(* IEC 61131-3 sources: Nauka-PLC-ST/ (part 2) *)

(* ---- Sterownik_Prasy_Formujacej.st ---- *)
VAR
    Start : BOOL;           // Przycisk monostabilny (musi być trzymany)
    Czujnik_detalu : BOOL;  // Potwierdzenie obecności materiału
    Czujnik_gora : BOOL;    // Czujnik prasy w gornym polozeniu
    Czujnik_dol : BOOL;     // Czujnik prasyw dolnym polozeniu
    Zawor_3_2 : BOOL;       // 1 - wysunięcie, 0 - schowanie (sprężyna)
    Krok_ukladu : INT := 0;
    Timer_prasowania : TON;
END_VAR

Timer_prasowania(PT := T#5S);

CASE Krok_ukladu OF
    0:  // IDLE - Czekamy na start i detal
        Zawor_3_2 := FALSE;
        Timer_prasowania.IN := FALSE;

        IF Start AND Czujnik_detalu THEN
            Krok_ukladu := 1;
        END_IF;

    1:  // ruch silownika w dol
        IF Start THEN
            Zawor_3_2 := TRUE;
            IF Czujnik_dol THEN // pzrechodzimy dopiero gdy silownik zjedzie na dol
                Krok_ukladu := 2;
            END_IF;
        ELSE
            // silownik wraca gdy puszcze przycisk start
            Krok_ukladu := 0;
        END_IF;

    2:  // czas pasowania detalu
        IF Start THEN
            Zawor_3_2 := TRUE;
            Timer_prasowania.IN := TRUE; // timer odlicza czas

            IF Timer_prasowania.Q THEN
                Krok_ukladu := 3;
            END_IF;
        ELSE
            Krok_ukladu := 0; // przerwanie prasowania
        END_IF;

    3:  // powrot silownika do stanu poczatkowego
        Zawor_3_2 := FALSE;
        Timer_prasowania.IN := FALSE;

        // Czekamy chwilę aż siłownik wróci (można dodać czujnik góra)
        IF NOT Start AND Czujnik_gora THEN
            Krok_ukladu := 0;
        END_IF;
END_CASE;

(* ---- Sterownik_przedmuchu_filtrow.st ---- *)
VAR
    Presostat_roznicy_p  : BOOL;  // czujnik przekroczenia max roznicy cisnien - filtr zapchany
    Zezwolenie_pracy     : BOOL;  // sygnal potwierdzajacy prace wlownego wentylatora

    Timer_impulsu        : TON;   // timer kontrolujacy czas trwania strzalu powietrza (np. 500ms)
    Timer_pauzy          : TON;   // timer liczacy przerwe miedzy strzalami roznych sekcji
    Krok                 : INT;   // krok ukladu: 0-spoczynek, 1-strzal 1, 2-pauza, 3-strzal 2

    Zawor_Przedmuchu_1   : BOOL;  // elektrozawor sprzonego powietrza dla sekcji 1
    Zawor_Przedmuchu_2   : BOOL;  // elektrozawor sprzonego powietrza dla sekcji 2
END_VAR

CASE Krok OF
    0: // Oczekiwanie na sygnal zapchania filtra przy pracy
        IF Presostat_roznicy_p AND Zezwolenie_pracy THEN
            Krok := 1; // rozpoczecie regeneracji
        END_IF;

    1: // strzal powietrza - sekcja 1
        IF Timer_impulsu.Q THEN
            Krok := 2; // koniec strzalu -> przejdz do pauzy
        END_IF;

    2: // przerwa na powrot cisnienia w zbiorniku
        IF Timer_pauzy.Q THEN
            Krok := 3; // powrot cisnienia -> strzal na sekcje 2
        END_IF;

    3: // Strzal powietrza - sekcja 2
        IF Timer_impulsu.Q THEN
            Krok := 0; // koniec oczyszczania -> powrot do czuwania
        END_IF;
END_CASE;

// timery
Timer_impulsu(IN := (Krok = 1) OR (Krok = 3), PT := T#500ms);  // czas pojedynczego strzalu powietrza

Timer_pauzy(IN := (Krok = 2), PT := T#4s);  // czas powrotu cisnienia

// sterowanie wyjsciami
Zawor_Przedmuchu_1 := Zezwolenie_pracy AND (Krok = 1);
Zawor_Przedmuchu_2 := Zezwolenie_pracy AND (Krok = 3);

(* ---- Sterownik_rozladunku_silosu.st ---- *)
VAR
    Zadanie_rozladunku   : BOOL;  // sygnal zadania startusekwencji programu
    Czujnik_przeplywu    : BOOL;  // czujnik lub fotokomorka wykrywajacy fizyczny zrzut materialu
    Krancowka_zasuwy     : BOOL;  // potwierdzenie pelnego otwarcia zasuwy pod silosem

    Timer_aeracji        : TON;   // czas trwania strzalu powietrza
    Timer_wibracji       : TON;   // czas pracy wibratora
    Krok                 : INT;   // krok sekwencji

    Zasuwa_nozowa        : BOOL;  // otwarcie zasuwy odcinajacej silos
    Zawor_aeracji        : BOOL;  // cewka elektrozaworu wtrysku powietrza
    Wibrator_stozka      : BOOL;  // stycznik silnika wibracyjnego na plaszczu
END_VAR

CASE Krok OF
    0: // stan czuwania - oczekiwanie na rozpoczecie sekwencji
        IF Zadanie_rozladunku THEN
            Krok := 1; // rozpoczecie rozladunku
        END_IF;

    1: // standardowy zrzut po otwarciu zrzutu
        IF NOT Zadanie_rozladunku THEN
            Krok := 0; // koniec rozladunku
        ELSIF Zadanie_rozladunku AND NOT Czujnik_przeplywu AND Krancowka_zasuwy THEN
            Krok := 2; // otawrta zasuwa - wykryto zwis
        END_IF;

    2: // spulchnianie materialu
        IF NOT Zadanie_rozladunku THEN
            Krok := 0;
        ELSIF Timer_aeracji.Q THEN
            IF Czujnik_przeplywu THEN
                Krok := 1; // powrot do standardowego zrzutu
            ELSE
                Krok := 3; // przejscie do wibracji
            END_IF;
        END_IF;

    3: // aktwyacja wibratora
        IF NOT Zadanie_rozladunku OR Timer_wibracji.Q OR Czujnik_przeplywu THEN
            Krok := 1; // powrot do oczekiwanie na rozpoczecie nowej sekwencji
        END_IF;
END_CASE;

// timer

Timer_aeracji(IN := (Krok = 2), PT := T#4s); // strzal powietrz trwa 4 sekundy

// Praca wibratora ograniczona do 3 sekund, aby chronic strukture mechaniczna i spawy silosu
Timer_wibracji(IN := (Krok = 3), PT := T#3s);

// sterowanie wyjsciami
Zasuwa_nozowa   := (Krok = 1) OR (Krok = 2) OR (Krok = 3);
Zawor_aeracji   := (Krok = 2);
Wibrator_stozka := (Krok = 3);

(* ---- Sterownik_stacji_obrotowej.st ---- *)
VAR
    Paleta_na_stacji     : BOOL;  // fotokomorka obecnosci palety na obrotnicy
    Krancowka_pozycja_0  : BOOL;  // czujnik pozycji bazowej 0 stopni
    Krancowka_pozycja_90 : BOOL;  // czujnik pozycji odwroconej  90 stopni
    Zgoda_na_wydanie     : BOOL;  // sygnal gotowosci na przyjecie palety

    Timer_stabilizacji   : TON;   // timer odliczajacy pelne zatrzymanie przed obrotem
    Krok                 : INT;   // krok sekwencji: 0-wejscie, 1-obrot_w_tok, 2-wydanie, 3-powrot

    Rolki_stacji_naprzod : BOOL;  // silnik rolek obrotnicy - ruch w przod
    Silnik_obrotu_90     : BOOL;  // silnik obracajacy stacje do pozycji 90 stopni
    Silnik_powrotu_0     : BOOL;  // silnik wracajacy stacje do pozycji 0 stopni
END_VAR

CASE Krok OF
    0: // oczekiwanie na palete w pozycji bazowej 0 stopni
        Rolki_stacji_naprzod := NOT Paleta_na_stacji AND Krancowka_pozycja_0;

        IF Paleta_na_stacji AND Krancowka_pozycja_0 AND Timer_stabilizacji.Q THEN
            Krok := 1; // paleta zajela stacje i zatrzymala sie -> start obrotu
        END_IF;

    1: // obrot stacji o 90 stopni do przenosnika
        IF Krancowka_pozycja_90 THEN
            Krok := 2; // osiagnieto pozycje 90 stopni -> przejscie do wydania
        END_IF;

    2: // wydanie palety na kolejny odcinek linii
        IF NOT Paleta_na_stacji THEN
            Krok := 3; // paleta opuscila stacje -> mozna wracac
        END_IF;

    3: // powrot obrotnicy do pozycji bazowej 0 stopni
        IF Krancowka_pozycja_0 THEN
            Krok := 0; // Stacja wrocila na pozycje startowa -> gotowa na nowa palete
        END_IF;
END_CASE;

// timery - 1,5 sekundy na zgaszenie sie drgan i zatrzymaniu po wjechaniu na stacje
Timer_stabilizacji(IN := Paleta_na_stacji AND Krancowka_pozycja_0, PT := T#1500ms);

// wyjscia
Silnik_obrotu_90     := (Krok = 1);
Rolki_stacji_naprzod := (Krok = 0 AND NOT Paleta_na_stacji) OR (Krok = 2 AND Zgoda_na_wydanie);
Silnik_powrotu_0     := (Krok = 3);

(* ---- Sterownik_windy_towarowej.st ---- *)
VAR
    Wezwanie_pietro_1    : BOOL;  // przycisk wezwania windy na pietro 1
    Wezwanie_pietro_2    : BOOL;  // przycisk wezwania windy na pietro 2
    Czujnik_pietro_1     : BOOL;  // czujnik krancowky obecnosci windy na pietrze 1
    Czujnik_pietro_2     : BOOL;  // czujnik krancowy obecnosci windy na pietrze 2
    Rygiel_zamkniety     : BOOL;  // czujnik bezpieczenstwa - drzwi zablokowane

    Timer_rygla          : TON;   // blokada bezpieczenstwa
    Krok                 : INT;   // krok ukladu: 0-stop, 1-ryglowanie, 2-ruch_w_gore, 3-ruch_w_dol

    Silnik_gora          : BOOL;  // stycznik poruszajacy winde w gore
    Silnik_dol           : BOOL;  // stycznik poruszajacy winde w dol
    Zwolnij_rygiel       : BOOL;  // cewka otwierajaca brzmi przy postoju
END_VAR

// sekwencja
CASE Krok OF
    0: // Stop - oczekiwanie na wezwanie windy na odpowiednie pietro
        IF Wezwanie_pietro_2 AND Czujnik_pietro_1 THEN
            Krok := 1; // Winda jest na dole, wezwano do gory -> ryglowanie drzwi
        ELSIF Wezwanie_pietro_1 AND Czujnik_pietro_2 THEN
            Krok := 1; // Winda jest na gorze, wezwano w dol -> ryglowanie drzwi
        END_IF;

    1: // sprawdzanie bezpieczenstwa przed startem silnika
        IF Rygiel_zamkniety AND Timer_rygla.Q THEN
            IF Wezwanie_pietro_2 THEN
                Krok := 2; // drzwi zablokowane bezpiecznie, ruch w gore
            ELSE
                Krok := 3; // drzwi zablokowane bezpiecznie, ruch w dol
            END_IF;
        ELSIF NOT Wezwanie_pietro_1 AND NOT Wezwanie_pietro_2 THEN
            Krok := 0; // reset kroku przy braku wezwania
        END_IF;

    2: // ruch w gore, winda jedzie na pietro 2
        IF Czujnik_pietro_2 OR NOT Rygiel_zamkniety THEN
            Krok := 0; // winda na miejscu lub przerwano rygiel, bezpieczny stop
        END_IF;

    3: // ruch w dol, winda jedzie na pietro 1
        IF Czujnik_pietro_1 OR NOT Rygiel_zamkniety THEN
            Krok := 0; // dojechano na miejsce lub przerwano rygiel, bezpieczny stop
        END_IF;
END_CASE;

// blokada bezpieczenstwa, timer odlicza 2 sek po ryglu aby wyeliminowac drgania stykow krancowek
Timer_rygla(IN := (Krok = 1) AND Rygiel_zamkniety, PT := T#2s);

(* ---- Sterownik_wozka_wahadlowego.st ---- *)
VAR
    Wozek_na_pozycji     : BOOL;  // czujnik gdy wozek stoi idealnie przed stacja
    Paczkowany_na_wozku  : BOOL;  // sygnal z fotokomorki potwierzdajacy obecnosc paczki
    Zadanie_zrzutu       : BOOL;  // sygnal nadrzedny dozkazujacy rozladunek paczki
    Sygnal_odbioru_stacji: BOOL;  // sygnal gotowosci do przejecia paczki

    Timer_transportera   : TON;   // timer czasu pracy wozka
    Krok                 : INT;   // krok sekwencji

    Rygluj_wozek         : BOOL;  // wygiel stabilizujacy wozek
    Uruchom_pas_wozka    : BOOL;  // tasma zamontowana na wozku
END_VAR

CASE Krok OF
    0: // wozek w ruchu lub czeka na sygnal
        IF Wozek_na_pozycji AND Paczkowany_na_wozku AND Zadanie_zrzutu THEN
            Krok := 1; // dojechal do celu - rygiel pozycjonujacy
        END_IF;

    1: //stabilizacja wozka do odbioru paczki
        IF NOT Wozek_na_pozycji THEN
            Krok := 0; // stop sekwencji gdy wozek sie przesunie
        ELSIF Sygnal_odbioru_stacji THEN
            Krok := 2; // gdy stacja gotowwa --> rozpocznij transfer
        END_IF;

    2: // rozladunek
        IF NOT Paczkowany_na_wozku AND Timer_transportera.Q THEN
            Krok := 3; // paczka opuscila wozek
        ELSIF NOT Wozek_na_pozycji THEN
            Krok := 0; // gdy dochodzido bledu pozycji to odetnij naped
        END_IF;

    3: // zakonczenie cyklu i odryglowanie wozka
        IF NOT Rygluj_wozek THEN
            Krok := 0; // wozek moze jechac dalej
        END_IF;
END_CASE;

// timery - pas pracuje 2 sekundy po braku sygnali z fotokomorki
Timer_transportera(IN := (Krok = 2) AND NOT Paczkowany_na_wozku, PT := T#2s);

// sterowaie wyjsciami
Rygluj_wozek      := (Krok = 1) OR (Krok = 2);
Uruchom_pas_wozka := (Krok = 2) AND Wozek_na_pozycji AND Sygnal_odbioru_stacji;

(* ---- Sterownik_zwrotnicy_sortujacej.st ---- *)
VAR
    Sygnal_odrzutu       : BOOL;  // sygnal z systemu wizyjnego dla detalu wadliwego
    Czujnik_pozycji      : BOOL;  // fotokomorka synchronizujaca na poczatku strefy sortowania
    Krancowka_silownika  : BOOL;  // czujnik wykrywajacy pelne cofniecie spychacza

    Timer_dolotu         : TON;   // timer czasu transportu paczki do miejsca zepchniecia
    Timer_wysuwu         : TON;   // timer okresu wysuwu silownika
    Krok                 : INT;   // krok sekwencji: 0-idle, 1-dolot, 2-spychanie, 3-powrot

    Silownik_odrzutu     : BOOL;  // cewka zaworu spychacza
END_VAR

CASE Krok OF
    0: // Czekanie na wadliwy detal i synchronizacje na fotokomorce
        IF Sygnal_odrzutu AND Czujnik_pozycji AND Krancowka_silownika THEN
            Krok := 1; // Detal wykryty, rozpoczecie liczenia czasu transportu
        END_IF;

    1: // Transport paczki przed silownik
        IF Timer_dolotu.Q THEN
            Krok := 2; // paczka na miejscu, uruchom spychacz
        END_IF;

    2: // Zepchniecie detalu
        IF Timer_wysuwu.Q THEN
            Krok := 3; // po okreslonym czasie, powrot spychacza
        END_IF;

    3: // Powrot silownika
        IF Krancowka_silownika THEN
            Krok := 0; // silownik schowany, oczekwianei na kolejny detal
        END_IF;
END_CASE;

// Timery
Timer_dolotu(IN := (Krok = 1), PT := T#2500ms);  // czas transportu paczki od fotokomorki do silownika

Timer_wysuwu(IN := (Krok = 2), PT := T#1s);  // silownik ma byc wysuniety przez 1 sekunde

// Sterowanie fizyczne
Silownik_odrzutu := (Krok = 2);

(* ---- System_nawadniania_szklarni.st ---- *)
VAR
Start : BOOL;  // przycisk uruchamiajacy system
Numer_sekcji : INT := 1;
Czas_podlewania : ARRAY[1..4] OF TIME := [T#10s, T#20s, T#25s, T#40s];
Zawory : ARRAY[1..4] OF BOOL;  // tablica wyjsc na kolejne zawory
Praca : BOOL;  // flaga pracy
Krok : INT := 0;  // numer kroku
Timer_podlewania : TON;  // timer czasu podlewania sekcji
END_VAR

IF Start THEN
Praca := 1;  // pamiec pracy ukladu
END_IF;

IF Praca Then
  Case Krok OF
  0:  // ustawienie sekcji
      Numer_sekcji := 1;
      Krok := 10;

  10:  // otwarcie odpowiedniego zaworu
      Zawory[Numer_sekcji] := TRUE;
      Timer_podlewania.PT := Czas_podlewania[Numer_sekcji];
      Timer_podlewania.IN := TRUE;  // start odliczania podlewania

      IF Timer_podlewania.Q THEN
          Krok := 20;
      END_IF;

  20:  // zamkniecie odpowiedniego zaworu i przejscie dalej
      Zawory[Numer_sekcji] := FALSE;
      Timer_podlewania.IN := FALSE;  // wylaczenie timera czasu podlewania

      // sekwencja przejscia do kolejnej sekcji
      IF Numer_sekcji < 4 THEN
        Numer_sekcji := Numer_sekcji + 1;
        Krok := 10;  // powrot i podlanie kolejnej sekcji
      ELSE
        Praca := FALSE;  // po podlaniu wszystkiego wylacz uklad
        Krok := 0;  // powrot do pierwszego kroku czekajacego na uruchomienie
      END_IF;
  END_CASE;

Timer_podlewania();

END_IF;

(* ---- System_obslugi_alarmow.st ---- *)
VAR
    bladCzujnika    : BOOL;   // czujnik PNP wykrywajacy blad czujnika
    bladPompy       : BOOL;   // czujnik PNP wykrywajacy blad pompy
    resetAlarmu     : BOOL;   // przycisk NC resetujacy calkowicie alarm

    Krok            : INT;    // Zapomniałeś o deklaracji zmiennej sterującej CASE
    lampkaAlarmu    : BOOL;   // lampka sygnalizuja alarm w ukladzie
    flagaAlarmu     : BOOL;   // pamiec wystapienia alarmu
    TON_swiecenie   : TON;    // czasowka do generatora impulsow - stan wysoki
    TON_przerwa     : TON;    // // czasowka do generatora impulsow - stan niski
END_VAR

// generator impulsow 1 Hz
TON_przerwa(IN := NOT TON_swiecenie.Q AND flagaAlarmu, PT := T#500MS);
TON_swiecenie(IN := TON_przerwa.Q, PT := T#500MS);

CASE Krok OF

  0:  // oczekiwanie na awarie
      IF bladCzujnika OR bladPompy THEN
        flagaAlarmu := TRUE;
        Krok := 1;
      END_IF;

  1: // sygnalizacja migajaca lampki
      lampkaAlarmu := TON_swiecenie.Q;

      IF NOT resetAlarmu THEN
        flagaAlarmu := FALSE; // wylaczenie migotania diody
        Krok := 2;
      END_IF;

  2: // potwierdzenie - lampka sygnalizacja jednostajna, czekanie na naprawienie awarii
      lampkaAlarmu := TRUE;

      IF NOT bladCzujnika AND NOT bladPompy THEN
        lampkaAlarmu := FALSE;
        Krok := 0; // powrot do stanu poczatkowego
      END_IF;

END_CASE;

(* ---- System_oddymiania_klatki.st ---- *)
VAR
    Sygnal_SAP          : BOOL;   // czujnik pozaru
    Przycisk_strazaka   : BOOL;   // reczny przycisk oddymiania
    Krancowka_klapy     : BOOL;   // krancowka klapy dymowej
    Czyste_powietrze    : BOOL;   // czujnik wykrywajacy czyste powietrze(brak dymu)
    Klapa_dymowa_otworz : BOOL;   // otwieranie klapy dymowej
    Wentylator_nawiew   : BOOL;   // wentylator podajacy powietrze
    Syrena_alarmowa     : BOOL;   // sygnal dzwiekowy
    Alarm_awaria_klapy  : BOOL;   // blad krytyczny otwierania klapy
    Timer_otwarcia      : TON;    // czas otwierania klapy
END_VAR

// procedura oddymiania
IF Sygnal_SAP OR Przycisk_Strazaka THEN
    Klapa_Dymowa_Otworz := TRUE;
    Syrena_Alarmowa     := TRUE;
ELSE
    Klapa_Dymowa_Otworz := FALSE;
    Syrena_Alarmowa     := FALSE;
END_IF;

// sterowanie wentylatora napowietrzajacego robiacy nadcisnienie gdy klapa jest otwarta
IF Klapa_Dymowa_Otworz AND Krancowka_Klapy AND Czyste_Powietrze_OK THEN
    Wentylator_Nawiew := TRUE;
ELSE
    Wentylator_Nawiew := FALSE;
END_IF;

// detekcja uszkodzenia, przy otwarciu mierzymy czas
Timer_Otwarcia(IN := Klapa_Dymowa_Otworz, PT := T#5S);

// jesli po czasie nie ma sygnalu z krancowki - ALARM
IF Timer_Otwarcia.Q AND NOT Krancowka_Klapy THEN
    Alarm_Awaria_Klapy := TRUE;
ELSE
    Alarm_Awaria_Klapy := FALSE;
END_IF;

(* ---- System_sortowania_paczek.st ---- *)
VAR
    Czujnik_obecnosci : BOOL;   // Wykrywa paczke na linii
    Czujnik_wagi : REAL;        // Waga paczki (0.0 - 10.0 kg)
    Silnik_tasmy : BOOL;        // Napęd głowny
    Spychacz_w_lewo : BOOL;     // Spycha lekkie paczki
    Spychacz_w_prawo : BOOL;    // Spycha ciezkie paczki

    Krok_ukladu : INT := 0;     // Stan ukladu
    Timer_Przejazd : TON;       // Timer odmierzajacy 2s dojazdu
END_VAR

// Wywołanie timera
Timer_przejazd(PT := T#2S);

// KROK 0: Oczekiwanie na paczkę
IF Krok_ukladu = 0 AND Czujnik_obecnosci THEN
    Silnik_tasmy := TRUE;
    Timer_przejazd.IN := TRUE; // Start odliczania
    Krok_ukladu := 1;
END_IF;

// KROK 1: Decyzja o sortowaniu (po minieciu 2 sekundach)
IF Krok_ukladu = 1 AND Timer_przejazd.Q THEN
    IF Czujnik_wagi < 5.0 THEN
        Spychacz_w_lewo := TRUE;
    ELSE
        Spychacz_w_prawo := TRUE;
    END_IF;
    Krok_ukladu := 2;
END_IF;

// KROK 2: Sprzątanie i powrót (paczka znika z czujnika)
IF Krok_ukladu = 2 AND NOT Czujnik_obecnosci THEN
    Silnik_tasmy := FALSE;
    Spychacz_w_lewo := FALSE;
    Spychacz_w_prawo := FALSE;
    Timer_przejazd.IN := FALSE; // Reset timera
    Krok_ukladu := 0;
END_IF;

(* ---- Tablica_pomiarow_filtr_cyfrowy.st ---- *)
VAR
    // Dane wejściowe
    Przeplyw_L_min : REAL;      // chwilowe zużycie
    ResetStatystyk : BOOL;      // przycisk zerujący

    // Logika tablicowa
    Historia_Zuzycia : ARRAY[0..9] OF REAL;
    LicznikTablicy : INT := 0;
    SredniaZuzycia : REAL;

    // Zmienne pomocnicze
    i : INT;                    // zmienna
    Suma_Pomocnicza : REAL;
    TimerZapisu : TON;          // deklaracja bloku czasowego

    // Diagnostyka
    AlarmPrzeciazenie : BOOL;
END_VAR

VAR_CONSTANT
    ProgSerwisowy : REAL := 8.5;
END_VAR

// cykliczny pomiar co 5 sekund
TimerZapisu(IN := NOT TimerZapisu.Q, PT := T#5S); // generator 5 sek

IF TimerZapisu.Q THEN
    // przesuniecie danych w tył tablicy
    FOR i := 9 TO 1 BY -1 DO
        Historia_Zuzycia[i] := Historia_Zuzycia[i-1];
    END_FOR;

    // wpisanie najnowszego pomiaru na początek
    Historia_Zuzycia[0] := Przeplyw_L_min;
END_IF;

// obliczenie sredniej średniej
Suma_Pomocnicza := 0.0;

FOR i := 0 TO 9 DO
    Suma_Pomocnicza := Suma_Pomocnicza + Historia_Zuzycia[i];
END_FOR;

SredniaZuzycia := Suma_Pomocnicza / 10.0;

// kontrola progu alarmowego
IF SredniaZuzycia > ProgSerwisowy THEN
    AlarmPrzeciazenie := TRUE;
ELSE
    AlarmPrzeciazenie := FALSE;
END_IF;

(* ---- Transporter_tasmowy.st ---- *)
VAR
    Tryb_pracy      : INT;     // 0-OFF, 1-AUTO, 2-SERVICE
    Czujnik_paczki  : BOOL;    // Fotokomorka
    Przycisk_jazdy  : BOOL;    // Dla trybu SERVICE (JOG)
    E_STOP          : BOOL;    // TRUE = OK, FALSE = ALARM
    Silnik_wyjscie  : BOOL;
    Licznik_total   : INT;

    Timer_jazdy     : TP;      // Timer impulsowy 5s
    R_Trig_licznik  : R_TRIG;
END_VAR

// --- WYWOŁANIE BLOKÓW (Zawsze na początku) ---
Timer_jazdy(IN := (Tryb_pracy = 1 AND Czujnik_paczki), PT := T#5S);
R_Trig_licznik(CLK := Silnik_wyjscie);

// --- 1. NADRZEDNE BEZPIECZENSTWO ---
IF NOT E_STOP THEN
    Tryb_pracy := 0;
END_IF;

// --- 2. AUTOMAT STANOW ---
CASE Tryb_pracy OF
    0: // STAN: OFF
        Silnik_wyjscie := FALSE;

        IF E_STOP THEN
            IF Czujnik_paczki THEN
                Tryb_pracy := 1; // Przejdz do AUTO
            ELSIF Przycisk_jazdy THEN
                Tryb_pracy := 2; // Przejdz do SERVICE
            END_IF;
        END_IF;

    1: // STAN: AUTO
        Silnik_wyjscie := Timer_jazdy.Q;

        // Powrot do OFF po zakonczeniu cyklu
        IF NOT Timer_jazdy.Q AND NOT Czujnik_paczki THEN
            Tryb_pracy := 0;
        END_IF;

    2: // STAN: SERVICE
        Silnik_wyjscie := Przycisk_jazdy;

        // Powrot do OFF, gdy operator pusci przycisk jazdy
        IF NOT Przycisk_jazdy THEN
            Tryb_pracy := 0;
        END_IF;
END_CASE;

// --- 3. LICZENIE PACZEK ---
IF R_Trig_licznik.Q THEN
    Licznik_total := Licznik_total + 1;
END_IF;

(* ---- Watchdog.st ---- *)
VAR
    Ping_OK          : BOOL;    // ptwierdzenie sygnalu z serwera TRUE = jest internet

    Timer_Brak_Ping  : TON;     // odliczanie czasu braku odpowiedzi
    Timer_Resetu     : TP;      // generator kontrolowanego impulsu odciecia zasilania
    Timer_Rozruchu   : TON;     // blokada sprawdzania pingu podczas uruchamiania routera

    Reset_Przekaznik : BOOL;    // Wyjście fizyczne odcinające zasilanie routera
END_VAR

Timer_Rozruchu(IN := NOT Reset_Przekaznik, PT := T#180s);    // sprawdza ping po 3 minutowym restarcie,

Timer_Brak_Ping(IN := NOT Ping_OK AND Timer_Rozruchu.Q, PT := T#60s);    // brak pingu ale tylko po zakonczeniu rozruchu

Timer_Resetu(IN := Timer_Brak_Ping.Q, PT := T#5s);   // odetnij zasilanie tylko an 5 sekund

Reset_Przekaznik := Timer_Resetu.Q;    // pokazanie sygnalu na sterowniku

(* ---- Winda_Magazynowa_Analogowa.st ---- *)
VAR
Pozycja_analog : INT;
Pozycja_zadana : INT;
Wybor_pietra : INT;
Obecne_pietro_windy : INT;
Waga : REAL;
Jazda_gora : BOOL;
Jazda_dol : BOOL;
Stop : BOOL;
Alarm_ukladu : BOOL;
Timer_pauzy : TON;
Przycisk_pietra_0 : BOOL;  //przycisk wyboru pietra 0
Przycisk_pietra_1 : BOOL;  //przycisk wyboru pietra 1
Przycisk_pietra_2 : BOOL;  //przycisk wyboru pietra 2
Przycisk_pietra_3 : BOOL;  //przycisk wyboru pietra 3
Przycisk_pietra_4 : BOOL;  //przycisk wyboru pietra 4
END_VAR;

IF Waga > 500 THEN  // wykrycie alarmu
Alarm_ukladu := TRUE;
END_IF;

Timer_pauzy(IN := (Przycisk_pietra_0 OR Przycisk_pietra_1 OR Przycisk_pietra_2 OR Przycisk_pietra_3 OR Przycisk_pietra_4)
  AND NOT Jazda_gora AND NOT Jazda_dol,
  PT := T#2s);

CASE Wybor_pietra OF
  0:  Pozycja_zadana := 0;
  1:  Pozycja_zadana := 250;
  2:  Pozycja_zadana :=500;
  3:  Pozycja_zadana := 750;
  4:  Pozycja_zadana := 1000;
END_CASE;

IF Przycisk_pietra_0 THEN
Wybor_pietra := 0;
END_IF;

IF Przycisk_pietra_1 THEN
Wybor_pietra := 1;
END_IF;

IF Przycisk_pietra_2 THEN
Wybor_pietra := 2;
END_IF;

IF Przycisk_pietra_3 THEN
Wybor_pietra := 3;
END_IF;

IF Przycisk_pietra_4 THEN
Wybor_pietra := 4;
END_IF;

IF Pozycja_analog > (Pozycja_zadana +10) AND Timer_pauzy.Q THEN  // jazda w DOL
Jazda_dol := TRUE;
Jazda_gora := FALSE;
END_IF;

IF Pozycja_analog < (Pozycja_zadana - 10) AND Timer_pauzy.Q THEN  // jazda w GORE
Jazda_gora := TRUE;
Jazda_dol := FALSE;
END_IF;

IF Pozycja_analog >= (Pozycja_zadana -10) AND Pozycja_analog <= (Pozycja_zadana + 10) THEN
Jazda_gora := FALSE;
Jazda_dol := FALSE;
END_IF;

IF Stop OR Alarm_ukladu THEN  // STOP LUB ALARM UKLADU
Jazda_dol := FALSE;
Jazda_gora := FALSE;
END_IF;

(* ---- Wykrywanie_poslizgu_tasmy.st ---- *)
VAR
    Impuls_bebna_napedu   : BOOL;  // czujnik obrotow napedu
    Impuls_rolki_zwrotnej : BOOL;  // czujnik obrotow rolki na koncu tasmy
    Silnik_tasmy_On       : BOOL;  // sygnal ze silnik w ogole powinien pracowac

    Licznik_napedu        : CTU;   // zliczanie impulsow z napedu
    Licznik_zwrotny       : CTU;   // zliczanie impulsow
    Timer_sprawdzania     : TON;   // weryfikacja poslizgu co 5 sekund

    Blokada_awaryjna      : BOOL;  // wykrycie poslizgu
END_VAR

// Zliczanie impulsów w pracy
Licznik_napedu(CU := Impuls_bebna_napedu, R := Timer_sprawdzania.Q OR NOT Silnik_tasmy_On);  // licznik zlicza zbocza narastajace z czujnika
Licznik_zwrotny(CU := Impuls_rolki_zwrotnej, R := Timer_sprawdzania.Q OR NOT Silnik_tasmy_On);  // licznik zwrotny zlicza jego obroty

// sprawdzanie roznicy co 5 sekund
Timer_sprawdzania(IN := Silnik_tasmy_On, PT := T#5s);  // okno pomiarowe

// bezpieczenstwo
IF Timer_sprawdzania.Q THEN  // sprawdza poslizg gdy minelo 5 sekund
    IF (Licznik_napedu.CV - Licznik_zwrotny.CV) >= 3 THEN  // sprawdza czy roznica obu licznikow wynosi wiecej niz 3
        Blokada_awaryjna := TRUE;  // jesli tasma ucieka lub zwalnia zalacz trwaly alarm
    END_IF;
END_IF;

(* ---- Zabezpieczenie_przeciwzamrożeniowe.st ---- *)
VAR
  tempNagrzewnicy : REAL;  // aktualna temperatura na powrocie wody z nagrzewnicy
  termostatBezpieczenstwa : BOOL;  // czujnik termostat bezpieczenstwa, TRUE jesli roznica temperatury powietrza a nagrzewnica spadnie ponizej 5 stopni
  wentNawiew : BOOL;  // sterowanie wentylatorem nawiewem
  zaworNagrzewnicy : BOOL;  // sterowanie zaworem nagrzewnicy
  alarm : BOOL;  // stan alarmu przeciwzamrozeniowego
END_VAR

IF (tempNagrzewnicy < 12.0) OR termostatBezpiecz THEN  // jesli niska temperatura wody lub sygnal z termostatu bezpieczenstwa
    alarm := TRUE;
END_IF;

IF (tempNagrzewnicy > 20.0) AND NOT termostatBezpiecz THEN  // warunek wylaczenia a - temp wody bezpeieczna i brak sygnalo z termostatBezpieczenstwa
    alarm := FALSE;
END_IF;

// co jesli jest alarm
IF alarm THEN
    wentNawiew      := FALSE; // wyłącz wentylator zeby nie bylo mrozu
    zaworNagrzewnicy := TRUE;  // otworz zawor aby ogrzac wymiennik
ELSE
    // urzadzenia pracuja w trybie normalnym jesli nie ma alarmu
    wentNawiew      := TRUE;
    zaworNagrzewnicy := FALSE;
END_IF;

(* ---- Zadajnik_predkosci.st ---- *)
VAR
    Przycisk_Plus : BOOL;  // Przycisk zwiekszajacy predkosc
    Przycisk_Minus : BOOL;  // Predkosc zmniejszajacy predkosc
    Wartosc_Zadana : REAL; // Zmienna do przechowywania zmiennosci
    Step : REAL := 0.5;    // Wartosc zmiany predkosci

    R_Trig_Plus : R_TRIG;  // Wykrycie klikniecia Plus, zabezpieczenie przed przytrzymaniem przycisku
    R_Trig_Minus : R_TRIG; // Wykrycie klikniecia minus, zabezpieczenie przed przytrzymaniem przycisku
END_VAR

// Wykrywamy kliknięcia - zbocze
R_Trig_Plus(CLK := Przycisk_Plus);
R_Trig_Minus(CLK := Przycisk_Minus);

// Faktyczne zwiększanie
IF R_Trig_Plus.Q AND Wartosc_Zadana < 100.0 THEN
    Wartosc_Zadana := Wartosc_Zadana + Step;
END_IF;

// Faktyczne zmniejszanie
IF R_Trig_Minus.Q AND Wartosc_Zadana > 0.0 THEN
    Wartosc_Zadana := Wartosc_Zadana - Step;
END_IF;

// Ochrona przed praca w nimozliwych zakresach - ponizej 0, ponad 100 procent
Wartosc_Zadana := LIMIT(0.0, Wartosc_Zadana, 100.0);
